FUNCTION_BLOCK Control (* Composite Function Block Type *)
  (* Standard: 61499-2 *)
  (* Version 0.0, 6/3/2016, Andrei, nxtControl GmbH, template *)
  PACKAGE Main;
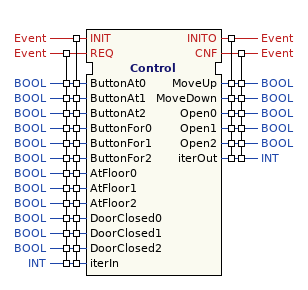
  EVENT_INPUT
    INIT WITH AtFloor0, AtFloor1, AtFloor2, DoorClosed0, DoorClosed1, DoorClosed2, ButtonAt0, ButtonAt1, ButtonAt2, ButtonFor0, ButtonFor1, ButtonFor2, iterIn; (* Initialization Request *)
    REQ WITH AtFloor0, AtFloor1, AtFloor2, DoorClosed0, DoorClosed1, DoorClosed2, ButtonAt0, ButtonAt1, ButtonAt2, ButtonFor0, ButtonFor1, ButtonFor2, iterIn; (* Normal Execution Request *)
  END_EVENT
  EVENT_OUTPUT
    INITO WITH MoveUp, MoveDown, Open0, Open1, Open2, iterOut; (* Initialization Confirm *)
    CNF WITH MoveUp, MoveDown, Open0, Open1, Open2, iterOut; (* Execution Confirmation *)
  END_EVENT
  VAR_INPUT
    ButtonAt0 : BOOL;
    ButtonAt1 : BOOL;
    ButtonAt2 : BOOL;
    ButtonFor0 : BOOL;
    ButtonFor1 : BOOL;
    ButtonFor2 : BOOL;
    AtFloor0 : BOOL;
    AtFloor1 : BOOL;
    AtFloor2 : BOOL;
    DoorClosed0 : BOOL;
    DoorClosed1 : BOOL;
    DoorClosed2 : BOOL;
    iterIn : INT;
  END_VAR
  VAR_OUTPUT
    MoveUp : BOOL; (* Output event qualifier *)
    MoveDown : BOOL;
    Open0 : BOOL;
    Open1 : BOOL;
    Open2 : BOOL;
    iterOut : INT;
  END_VAR
  FBS
    FB1 : DummyControl;
  END_FBS
  EVENT_CONNECTIONS
    REQ TO FB1.REQ;
    INIT TO FB1.INIT;
    FB1.INITO TO INITO;
    FB1.CNF TO CNF;
  END_CONNECTIONS
  DATA_CONNECTIONS
    AtFloor0 TO FB1.AtFloor0;
    AtFloor2 TO FB1.AtFloor2;
    AtFloor1 TO FB1.AtFloor1;
    DoorClosed0 TO FB1.DoorClosed0;
    DoorClosed1 TO FB1.DoorClosed1;
    DoorClosed2 TO FB1.DoorClosed2;
    ButtonAt0 TO FB1.Button0;
    ButtonAt1 TO FB1.Button1;
    ButtonAt2 TO FB1.Button2;
    ButtonFor0 TO FB1.Req0;
    ButtonFor1 TO FB1.Req1;
    ButtonFor2 TO FB1.Req2;
    FB1.liftUp TO MoveUp;
    FB1.liftDown TO MoveDown;
    FB1.door0 TO Open0;
    FB1.door1 TO Open1;
    FB1.door2 TO Open2;
  END_CONNECTIONS
END_FUNCTION_BLOCK
